FUNCTION_BLOCK PNP_PLANT_MS_CONTROL_FOR_SMV (* Composite Function Block Type *)
  (* Standard: 61499-2 *)
  (* Version 0.2, 2003-12-05, JHC, Rockwell Automation, Renamed from NEWCOMPFB. *)
  (* Version 0.1, 2002-01-08, JHC, Rockwell Automation, Added DLY FB as example. *)
  (* Version 0.0, 2000-05-27, JHC, Rockwell Automation *)
  (* Compiler header: package fb.rt.pnp; *)
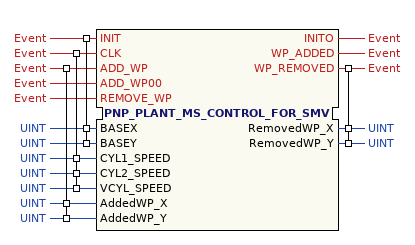
  EVENT_INPUT
    INIT WITH BASEX, BASEY; (* Initialisation *)
    CLK WITH CYL1_SPEED, CYL2_SPEED, VCYL_SPEED;
    ADD_WP WITH AddedWP_X, AddedWP_Y;
    ADD_WP00;
    REMOVE_WP;
  END_EVENT
  EVENT_OUTPUT
    INITO; (* Initialization Confirm *)
    WP_ADDED;
    WP_REMOVED WITH RemovedWP_X, RemovedWP_Y;
  END_EVENT
  VAR_INPUT
    BASEX : UINT;
    BASEY : UINT;
    CYL1_SPEED : UINT;
    CYL2_SPEED : UINT;
    VCYL_SPEED : UINT;
    AddedWP_X : UINT;
    AddedWP_Y : UINT;
  END_VAR
  VAR_OUTPUT
    RemovedWP_X : UINT;
    RemovedWP_Y : UINT;
  END_VAR
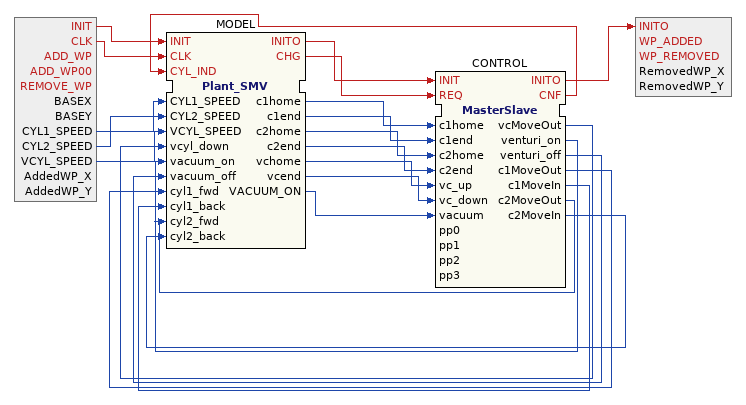
  FBS
    MODEL : Plant_SMV;
    CONTROL : MasterSlave;
  END_FBS
  EVENT_CONNECTIONS
    INIT TO MODEL.INIT;
    CLK TO MODEL.CLK;
    MODEL.INITO TO CONTROL.INIT;
    MODEL.CHG TO CONTROL.REQ;
    CONTROL.INITO TO INITO;
    CONTROL.CNF TO MODEL.CYL_IND;
  END_CONNECTIONS
  DATA_CONNECTIONS
    CYL1_SPEED TO MODEL.CYL1_SPEED;
    CYL2_SPEED TO MODEL.CYL2_SPEED;
    VCYL_SPEED TO MODEL.VCYL_SPEED;
    MODEL.c1home TO CONTROL.c1home;
    MODEL.c1end TO CONTROL.c1end;
    MODEL.c2home TO CONTROL.c2home;
    MODEL.c2end TO CONTROL.c2end;
    MODEL.vchome TO CONTROL.vc_up;
    MODEL.vcend TO CONTROL.vc_down;
    MODEL.VACUUM_ON TO CONTROL.vacuum;
    CONTROL.vcMoveOut TO MODEL.vcyl_down;
    CONTROL.venturi_on TO MODEL.vacuum_on;
    CONTROL.venturi_off TO MODEL.vacuum_off;
    CONTROL.c1MoveOut TO MODEL.cyl1_fwd;
    CONTROL.c1MoveIn TO MODEL.cyl1_back;
    CONTROL.c2MoveOut TO MODEL.cyl2_fwd;
    CONTROL.c2MoveIn TO MODEL.cyl2_back;
  END_CONNECTIONS
END_FUNCTION_BLOCK
